- Модуль ВЧ-демпфування: Несправність: перенапруга 24 В'; 37052 'F37052 - Модуль ВЧ-демпфування: Помилка даних EEPROM'; 37056 'A37056 (F) - Модуль ВЧ-демпфування: Перегрів радіатора'; 37310 'A37310 (F) - Модуль ВЧ-дроселя: Перегрів'; 37311 'F37311 - Модуль ВЧ-дроселя: Перегрів радіатора'; 37312 'A37312 (F) - Модуль ВЧ-дроселя: Перегрів або несправність вентилятора'; 37313 'F37313 - Модуль ВЧ-дроселя: Перегрів або несправність вентилятора'; 37502 'A37502 (F) - Модуль ВЧ-демпфування: Напруга демпфування занадто висока'; 37800 'N37800 (F) - Модуль ВЧ-демпфування: Груповий сигнал'; 37801 'A37801 (F, N) - Модуль ВЧ-демпфування: Відсутній сигнал справності'; 37802 'F37802 (N, A) - Модуль ВЧ-демпфування: Переповнення часового кванта'; 37804 'F37804 (N, A) - Модуль ВЧ-демпфування: CRC'; 37805 'F37805 - Модуль ВЧ-демпфування: Некоректна контрольна сума EEPROM'; 37820 'F37820 - Модуль ВЧ-демпфування: Помилка телеграми'; 37835 'F37835 - Модуль ВЧ-демпфування: Помилка циклічної передачі даних'; 37836 'F37836 - Модуль ВЧ-демпфування: Помилка передавання даних DRIVE-CLiQ'; 37837 'F37837 - Модуль ВЧ-демпфування: Несправність компонента'; 37845 'F37845 - Модуль ВЧ-демпфування: Помилка циклічної передачі даних'; 37850 'F37850 - Модуль ВЧ-демпфування: Внутрішня програмна помилка'; 37851 'F37851 - Модуль ВЧ-демпфування (CU): Відсутній сигнал справності'; 37860 'F37860 - Модуль ВЧ-демпфування (CU): Помилка телеграми'; 37875 'F37875 - Модуль ВЧ-демпфування: Несправність напруги живлення'; 37885 'F37885 - Модуль ВЧ-демпфування (CU): Помилка циклічної передачі даних'; 37886 'F37886 - Модуль ВЧ-демпфування (CU): Помилка під час передавання даних DRIVE-CLiQ'; 37887 'F37887 - Модуль ВЧ-демпфування (CU): Несправність компонента'; 37895 'F37895 - Модуль ВЧ-демпфування (CU): Помилка почергової циклічної передачі даних'; 37896 'F37896 - Модуль ВЧ-демпфування (CU): Некоректні властивості компонента'; 37899 'F37899 (N, A) - Модуль ВЧ-демпфування: Невідома несправність'; 37903 'F37903 - Модуль ВЧ-демпфування: Виникла помилка I2C-шини'; 37950 'F37950 - Модуль ВЧ-демпфування: Внутрішня програмна помилка'; 37999 'A37999 (F, N) - Модуль ВЧ-демпфування: Невідоме аварійне повідомлення'; 40000 'F40000 - Несправність роз’єму DRIVE-CLiQ X100'; 40001 'F40001 - Несправність роз’єму DRIVE-CLiQ X101'; 40002 'F40002 - Несправність роз’єму DRIVE-CLiQ X102'; 40003 'F40003 - Несправність роз’єму DRIVE-CLiQ X103'; 40004 'F40004 - Несправність роз’єму DRIVE-CLiQ X104'; 40005 'F40005 - Несправність роз’єму DRIVE-CLiQ X105'; 40100 'A40100 - Аварійне повідомлення роз’єму DRIVE-CLiQ X100'; 40101 'A40101 - Аварійне повідомлення роз’єму DRIVE-CLiQ X101'; 40102 'A40102 - Аварійне повідомлення роз’єму DRIVE-CLiQ X102'; 40103 'A40103 - Аварійне повідомлення роз’єму DRIVE-CLiQ X103'; 40104 'A40104 - Аварійне повідомлення роз’єму DRIVE-CLiQ X104'; 40105 'A40105 - Аварійне повідомлення роз’єму DRIVE-CLiQ X105'; 40799 'F40799 - CX32: Перевищено налаштований час завершення передавання'; 40801 'F40801 - CX32 DRIVE-CLiQ: відсутній сигнал справності'; 40820 'F40820 - CX32 DRIVE-CLiQ: помилка телеграми'; 40825 'F40825 - CX32 DRIVE-CLiQ: Несправність напруги живлення'; 40835 'F40835 - CX32 DRIVE-CLiQ: помилка циклічної передачі даних'; 40836 'F40836 - CX32 DRIVE-CLiQ: помилка передавання даних DRIVE-CLiQ'; 40837 'F40837 - CX32 DRIVE-CLiQ: несправність компонента'; 40845 'F40845 - CX32 DRIVE-CLiQ: помилка циклічної передачі даних'; 40851 'F40851 - CX32 DRIVE-CLiQ (CU): відсутній сигнал справності'; 40860 'F40860 - CX32 DRIVE-CLiQ (CU): помилка телеграми'; 40875 'F40875 - CX32 DRIVE-CLiQ (CU): Несправність напруги живлення'; 40885 'F40885 - CX32 DRIVE-CLiQ (CU): помилка циклічної передачі даних'; 40886 'F40886 - CX32 DRIVE-CLiQ (CU): помилка під час передавання даних DRIVE-CLiQ'; 40887 'F40887 - CX32 DRIVE-CLiQ (CU): несправність компонента'; 40895 'F40895 - CX32 DRIVE-CLiQ (CU): помилка циклічної передачі даних'; 49150 'F49150 - Охолоджувальний агрегат: Виникла несправність'; 49151 'F49151 - Охолоджувальний агрегат: Провідність перевищила поріг несправності'; 49152 'F49152 - Охолоджувальний агрегат: Відсутній сигнал зворотного зв’язку команди ON'; 49153 'F49153 - Охолоджувальний агрегат: Витрата рідини занадто мала'; 49154 'F49154 (A) - Охолоджувальний агрегат: Виявлено витік рідини'; 49155 'F49155 - Охолоджувальний агрегат: Адаптер Power Stack: версія прошивки застаріла'; 49156 'F49156 - Охолоджувальний агрегат: Температура охолоджувальної рідини перевищила поріг несправності'; 49170 'A49170 - Охолоджувальний агрегат: Виникло аварійне повідомлення'; 49171 'A49171 (N) - Охолоджувальний агрегат: Провідність перевищила поріг аварійного повідомлення'; 49172 'A49172 - Охолоджувальний агрегат: Фактичне значення провідності некоректне'; 49173 'A49173 - Охолоджувальний агрегат: Температура охолоджувальної рідини перевищила поріг аварійного повідомлення'; 49200 'F49200 - Несправність групового сигналу збудження'; 49201 'A49201 (F) - Аварійне повідомлення групового сигналу збудження'; 49204 'A49204 (N) - Аварійне повідомлення про вимкнення збудження'; 49205 'A49205 - Збудження: некоректна параметризація безщіткового збуджувача'; 49920 'A49920 (F) - Спрацював захисний автомат головного кола'; 49921 'A49921 (F) - Спрацював захисний автомат резервного головного кола'; 49922 'A49922 (F) - Спрацював захисний автомат кола 24 В'; 49923 'A49923 (F) - Спрацював захисний автомат кола 24 В клемної колодки'; 49924 'A49924 (F) - Спрацював захисний автомат кола живлення силового модуля'; 49926 'A49926 (F) - Спрацював захисний автомат кола синхронізувальної напруги'; 49927 'A49927 (F) - Спрацював захисний автомат кола допоміжного вентилятора'; 49933 'A49933 (F) - Спрацював захисний автомат кола збудження 230 В AC'; 49934 'A49934 (F) - Спрацював захисний автомат вихідного кола охолоджувального агрегату 230 В AC'; 49935 'A49935 (F) - Спрацював захисний автомат кола 24 В соленоїдів дверей силового модуля'; 49936 'A49936 - Спрацював захисний автомат кола освітлення/розеток 230 В AC'; 49937 'A49937 (F) - UPS не готовий до роботи'; 49938 'A49938 (F) - Робота від батареї UPS'; 49939 'A49939 (F) - Батарею UPS розряджено'; 49940 'A49940 (F) - Спрацював захисний автомат кола живлення силового модуля 400 В'; 49941 'A49941 (F) - Спрацював захисний автомат антиконденсаційного обігріву'; 49942 'A49942 (F) - Спрацював захисний автомат кола живлення SITOP'; 49998 'A49998 - Виникла подія запуску реєстратора'; 50002 'A50002 (F) - COMM BOARD: аварійне повідомлення 2'; 50003 'A50003 (F) - COMM BOARD: аварійне повідомлення 3'; 50004 'A50004 (F) - COMM BOARD: аварійне повідомлення 4'; 50005 'A50005 (F) - COMM BOARD: аварійне повідомлення 5'; 50006 'A50006 (F) - COMM BOARD: аварійне повідомлення 6'; 50007 'A50007 (F) - COMM BOARD: аварійне повідомлення 7'; 50008 'A50008 (F) - COMM BOARD: аварійне повідомлення 8'; 50011 'A50011 (F) - EtherNetIP/COMM BOARD: помилка конфігурації'; 0 'Немає помилки'

text list "PresetStatus": 0 'Немає помилки'; 32801 'Пресет заблоковано'; 33282 'Немає дозволу `PresetPermit`'; 33283 'Енкодер не готовий або є помилка комунікації'; 33284 'Preset вже активний.'; 33285 'Значення пресет поза допустимим діапазоном'

text list "EncoderStatus": 1 'Помилка читання'; 2 'Помилка запису'; 4 'Помилка комунікації'; 8 'Керування з ПЛК не активне'; 16 'Помилка енкодера'; 32 'Попередження енкодеру'; 256 'Sign-of-life енкодера не валідний'; 512 'Положення енкодера не достовірне'; 1024 'Швидкість енкодера не достовірна'; 2048 'Енкодер не готовий для використання в логіці'; 4096 'Симуляція енкодера актвина'; 8192 'Preset-процедура активна'; 8193 'Помилка виконання preset'

text list "StatusCodeCU320": 0 'Читання telegram CU → PLC виконано без помилки'; 1 'Запис telegram PLC → CU виконано без помилки'; 2 'Обмін з CU справний'; 3 'CU повідомляє fault'; 4 'CU повідомляє warning'; 5 'CU повідомляє заборону / блокування'; 6 'CU запитує керування від PLC'; 7 'Активний режим симуляції'

text list "StatusCodeDrive": 0 'Читання telegram ПЧ → PLC виконано без помилки'; 1 'Запис telegram PLC → ПЧ виконано без помилки'; 2 'ПЧ увімкнений та робота дозволена'; 3 'ПЧ не готовий до роботи або активна заборона / блокування'; 4 'Є аварія ПЧ'; 5 'Є попередження ПЧ'; 6 'ПЧ запитує відкриття гальма'; 7 'Активний режим симуляції'; 8 'Активна заборона вмикання'; 9 'ПЧ запитує керування від PLC'

